// TIA Portal V20 export
TYPE "typeSequenceControlNodeHomeCheck_topTapeFixStage"
// stored: Namespace Unit1.Em3
   STRUCT
      partNoDetect { ExternalWritable := 'False'} : Bool;
      partDetect { ExternalWritable := 'False'} : Bool;
   END_STRUCT;
END_TYPE
